// TIA Portal V19 export
TYPE "UDT_SIM_BOOL"
   STRUCT
      en : Bool;
      value : Bool;
   END_STRUCT;
END_TYPE
